// TwinCAT 3 PLC project PizzaOvenPLC
// ProgramVersion: 3.1.4022.1
// libraries:
//   Tc2_System, * (Beckhoff Automation GmbH)
//   Tc3_Module, * (Beckhoff Automation GmbH)
//   Tc2_Standard,3.3.2.0,Beckhoff Automation GmbH
//   Tc2_System,3.4.17.0,Beckhoff Automation GmbH
//   Tc3_Module,3.3.17.0,Beckhoff Automation GmbH
//   Visu Interfaces,3.5.5.0,System
// project tree:
//   DUTs/ ST_PIZZA.TcDUT
//   / GlobalTextList.TcGTLO, PlcTask.TcTTO, Visualization Manager.TcVMO (not stored)
//   POUs/ BrandAlarm.TcPOU, MAIN.TcPOU, FB_PIZZA_OVEN.TcPOU
//   VISUs/ ITF.TcIO, OvenHMI.TcVIS

CONFIGURATION PizzaOvenPLC
    RESOURCE PLC ON TwinCAT3
        TASK PlcTask(INTERVAL := T#10ms, PRIORITY := 20);
        PROGRAM MAIN WITH PlcTask : MAIN;
    END_RESOURCE
END_CONFIGURATION

// ---- DUTs/ST_PIZZA.TcDUT
TYPE ST_PIZZA :
STRUCT
END_STRUCT
END_TYPE

// ---- VISUs/ITF.TcIO
INTERFACE ITF

END_INTERFACE

// ---- POUs/MAIN.TcPOU
PROGRAM MAIN
VAR_INPUT
	
	Pizza_in 	: 				BOOL; 	//sensorlicht am eingang bricht ab, Teig is aufgeladen
	Pizza_out 	:				BOOL;  // Pizza entfernen
END_VAR
VAR
		i 			: 			DINT;
	//fbTrigEin		: 			R_TRIG;
	//Objeckt deklaration von class FB_Pizza_Oven
	veggie			: 			FB_PIZZA_OVEN; 
	salami			:			FB_PIZZA_OVEN;
//	p:							BrandAlarm;
END_VAR


CASE i+1 OF 
1:

veggie.PizzaEin:=pizza_in;				// Teig auf Förderbahn1
veggie.KochZeit:=T#3S;					// Kochzeit für Veggie pizza ist 3sekunden
veggie.PizzaAus:=pizza_out;				//pizza am Fließband wird entfernt
veggie.MethodPizza();

2:

salami.PizzaEin:=pizza_in;
salami.KochZeit:=T#7S;
salami.PizzaAus:=pizza_out;
salami.MethodPizza();

END_CASE

END_PROGRAM

// ---- POUs/FB_PIZZA_OVEN.TcPOU
	FUNCTION_BLOCK FB_PIZZA_OVEN 
VAR_INPUT
	Pizza_in 	: 			BOOL:=FALSE;
	Pizza_out 	:			BOOL:=FALSE;

	fbTrig		: 			R_TRIG;
	fbTrig2		: 			R_TRIG;
END_VAR

VAR_OUTPUT
	PizzaStatus	: 			STRING;
END_VAR
VAR
	_pizza_aus: 			BOOL;
	_pizza_ein:				BOOL;
	_brand_alarm: 			BOOL;
	_cook_time:				TIME;
		_count	:			DINT;
	
	fbTimer		: 			TON;
	fbTimer1	:			TON;
	
	_pizza_backen:			BOOL;
	
	_teig_auflade:			BOOL;

	_zutaten		:		BOOL;

	_pizza_fertig:			BOOL;
	_led_anzeige:			BOOL;

	iState		:  			DINT:=0;
	
END_VAR

PROPERTY BrandAlarm : BOOL
GET
BrandAlarm:=_brand_alarm;
END_GET
SET
_brand_alarm:=BrandAlarm;
END_SET
END_PROPERTY

PROPERTY IngridientDeck : BOOL
GET
IngridientDeck:=_zutaten;
END_GET
SET
_zutaten:=IngridientDeck;
END_SET
END_PROPERTY

PROPERTY KochZeit : TIME
GET
KochZeit:=_cook_time;
END_GET
SET
_cook_time:=KochZeit;
END_SET
END_PROPERTY

PROPERTY LedAnzeige : BOOL
GET
LedAnzeige:= _led_anzeige;
END_GET
SET
_led_anzeige:= LedAnzeige;
END_SET
END_PROPERTY

METHOD MethodBrandAlarm : BOOL
VAR_INPUT
END_VAR
END_METHOD

METHOD MethodCounter : DINT
VAR_INPUT
END_VAR
_count:=_count+1;
END_METHOD

METHOD MethodLedAnzeige : BOOL
VAR_INPUT
END_VAR

_led_anzeige:=TRUE;
END_METHOD

METHOD PUBLIC MethodPizza : UDINT
VAR


END_VAR
//control buttons
THIS^.MethodPizzaAufladen();
THIS^.MethodRemovePizza();
//status changes
CASE iState OF 
0:	PizzaStatus:='Offen Frei';
IF _teig_auflade AND NOT _zutaten THEN		
		_teig_auflade:=FALSE;
		_zutaten:=TRUE;
END_IF
fbTimer1(IN:=_zutaten,PT:=T#3S);
IF fbTimer1.Q THEN
	iState:=7;
END_IF 	
7: IF _zutaten AND NOT _pizza_backen THEN
					
		_zutaten:=FALSE;
		_pizza_backen:=TRUE;
		iState:=10;
END_IF
10:	IF _pizza_backen THEN
	  PizzaStatus:='Öffen besetzt...';
	THIS^.MethodLedAnzeige();
END_IF
	fbTimer(IN:=_pizza_backen,PT:=KochZeit);
IF fbTimer.Q THEN
	//PizzaInOven:=FALSE;
	THIS^.MethodCounter();
	iState:=20;
	
END_IF
	
20:	PizzaStatus:='Entladen';
IF  NOT _pizza_fertig THEN
	_brand_alarm:=FALSE;
	_pizza_backen:=FALSE;
	_pizza_fertig:=TRUE;
	fbTimer(IN:=FALSE);
	iState:=0;
	ELSE
		_brand_alarm:=TRUE;
	END_IF
	
END_CASE
END_METHOD

METHOD MethodPizzaAufladen : BOOL
VAR_INPUT
END_VAR
		fbTrig(CLK:=_pizza_ein);//load pizza button clicked trggered
IF		fbTrig.Q THEN		//When Triggerd 
		_teig_auflade:=TRUE;	
			iState:=0;
		//Pizza_in:=FALSE;
		//fbTrig(clk:=FALSE);
END_IF
END_METHOD

METHOD MethodRemovePizza : BOOL
VAR_INPUT
END_VAR
	fbTrig2(CLK:=_pizza_aus); 
IF 	fbTrig2.Q THEN
	_pizza_fertig:=FALSE;
	//Pizza_out:=FALSE;
	//fbTrig2(clk:=Pizza_out);
END_IF
END_METHOD

PROPERTY PizzaAus : BOOL
GET
PizzaAus:=_pizza_aus;
END_GET
SET
_pizza_aus:=PizzaAus;
END_SET
END_PROPERTY

PROPERTY PizzaDone : BOOL
GET
PizzaDone:=_pizza_fertig;
END_GET
SET
_pizza_fertig:=PizzaDone;
END_SET
END_PROPERTY

PROPERTY PizzaEin : BOOL
GET
PizzaEin:=_pizza_ein;
END_GET
SET
_pizza_ein:=PizzaEin;
END_SET
END_PROPERTY

PROPERTY PizzaInOven : BOOL
GET
PizzaInOven:=_pizza_backen;
END_GET
SET
_pizza_backen:=PizzaInOven;
END_SET
END_PROPERTY

PROPERTY PizzaOnDeck : BOOL
GET
PizzaOnDeck:=_teig_auflade;
END_GET
SET
_teig_auflade:=PizzaOnDeck;
END_SET
END_PROPERTY

PROPERTY Zaehler : DINT
GET
Zaehler:=_count;
END_GET
SET
_count:=Zaehler;
END_SET
END_PROPERTY

END_FUNCTION_BLOCK

// ---- POUs/BrandAlarm.TcPOU
FUNCTION_BLOCK BrandAlarm EXTENDS FB_PIZZA_OVEN
VAR_INPUT
	
END_VAR
VAR_OUTPUT
END_VAR
VAR
END_VAR

PROPERTY BrandAlarm : BOOL
GET
BrandAlarm:=_brand_alarm;
END_GET
SET
_brand_alarm:=BrandAlarm;
END_SET
END_PROPERTY

METHOD MethodSetAlarm : BOOL
VAR_INPUT
END_VAR
IF _pizza_fertig AND _pizza_backen THEN
_brand_alarm:=TRUE;
END_IF
END_METHOD

END_FUNCTION_BLOCK

// ---- GlobalTextList.TcGTLO
TEXTLIST GlobalTextList
  866 = '%d'
  852 = '%i'
  563 = '%s'
  89 = '%S'
  450 = '%t'
  901 = 'Backofen'
  304 = 'Fließband'
  556 = 'Förderbahn 1'
  478 = 'Förderbahn 2'
  742 = 'In Oven'
  596 = 'Insert Pizza'
  501 = 'Insert Pizza2'
  321 = 'Margaretha'
  751 = 'PizzaDone'
  181 = 'PizzaInOven'
  953 = 'Pizza_In'
  936 = 'Remove Pizza'
  815 = 'Salami'
  895 = 'Sauce'
  653 = 'Status: %s'
  297 = 'Status:%s'
  302 = 'Tomatenmark'
  61 = 'Veggie'
  217 = 'Zähler'
END_TEXTLIST

// ---- VISUs/OvenHMI.TcVIS
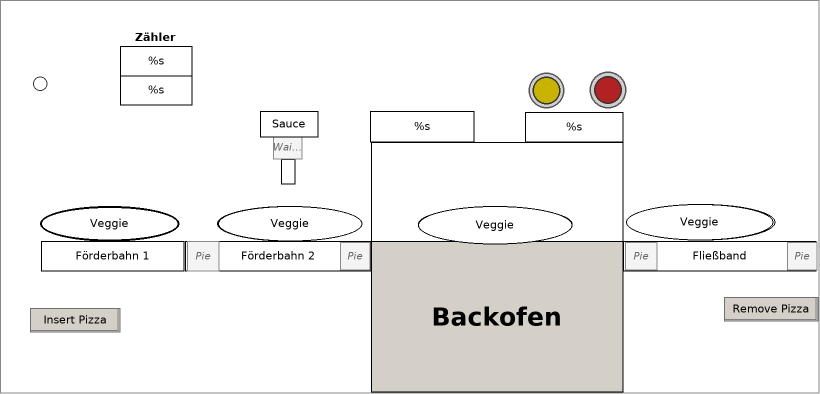
VISUALIZATION OvenHMI  // 820x394
    Rectangle (281,159 14x25), colour toggle: MAIN.veggie._zutaten MAIN.salami._zutaten
    Rectangle (185,241 186x30), "Förderbahn 2"
    Ellipse (217,206 143x35), "Salami", invisible if: NOT MAIN.salami._zutaten
    Rectangle (371,142 252x250)
    Rectangle (623,241 193x30), "Fließband"
    Ellipse (628,204 147x36), "Salami", invisible if: NOT MAIN.salami._pizza_fertig
    Button (30,308 90x24), "Insert Pizza"
        tap MAIN.Pizza_in
        OnMouseClick: execute {  }
    Button (724,297 94x24), "Remove Pizza"
        tap MAIN.Pizza_out
        OnMouseClick: execute {  }
    Ellipse (418,207 154x33), "Salami", invisible if: NOT MAIN.salami._pizza_backen
    Rectangle (371,241 252x151), "Backofen", colour toggle: MAIN.veggie._pizza_backen OR MAIN.salami._pizza_backen
    Pie (187,241 32x30)
    Pie (340,242 30x28)
    Pie (625,242 32x28)
    Pie (787,242 30x28)
    RadioButton (31,47 136x73), variable: MAIN.i
        Areas[0]: Text=Veggie
        Areas[1]: Text=Salami
    Ellipse (218,206 144x35), "Veggie", invisible if: NOT MAIN.veggie._zutaten
    Ellipse (418,206 154x38), "Veggie", invisible if: NOT MAIN.veggie._pizza_backen
    Ellipse (626,204 147x36), "Veggie", invisible if: NOT MAIN.veggie._pizza_fertig
    Rectangle (525,112 98x30), "%s", text variable: MAIN.salami.PizzaStatus, invisible if: MAIN.i=0
    Rectangle (371,112 103x30), "%s", text variable: MAIN.salami.fbTimer.ET, invisible if: MAIN.i=0
    Rectangle (120,75 72x30), "%s", text variable: MAIN.salami._count
    Rectangle (120,46 72x30), "%s", text variable: MAIN.veggie._count
    Rectangle (370,111 104x31), "%s", text variable: MAIN.veggie.fbTimer.ET, invisible if: MAIN.i=1
    Rectangle (525,112 98x30), "%s", text variable: MAIN.veggie.PizzaStatus, invisible if: MAIN.i=1
    Rectangle (41,241 143x30), "Förderbahn 1"
    Ellipse (40,206 139x35), "Salami", invisible if: NOT MAIN.salami._teig_auflade
    Lamp1 (524,70 45x41), variable: MAIN.salami._pizza_backen OR MAIN.veggie._pizza_backen, style: Lamp-Lamp1-Yellow
    Lamp1 (585,69 46x42), variable: MAIN.salami._brand_alarm OR MAIN.veggie._brand_alarm, style: Lamp-Lamp1-Red
    Ellipse (41,207 137x33), "Veggie", invisible if: NOT MAIN.veggie._teig_auflade
    WaitingSymbolFlower (273,135 29x24)
    Label (107,28 97x19), "Zähler"
    Rectangle (260,111 58x26), "Sauce"
END_VISUALIZATION
